PROGRAM MAIN
VAR
	xSwitch			: BOOL;
	xLamp	AT %Q*	: BOOL;
	
	astServoIF		: ARRAY[0..gc.usiMaxNrOfAxes] OF typ_ServoIF;
END_VAR

xLamp	:= xSwitch;

END_PROGRAM

(* stored: Version 1.1.0.1, ProductVersion 3.1.4022.17
   POU MAIN: Id {326ec9f8-804c-4728-ab87-9b4e7fbd17cf}, SpecialFunc None *)
